// Mitsubishi GX Works2 project: fx2N_may1truc_v1.0   PLC: FX2N/FX2NC

PROGRAM MAIN
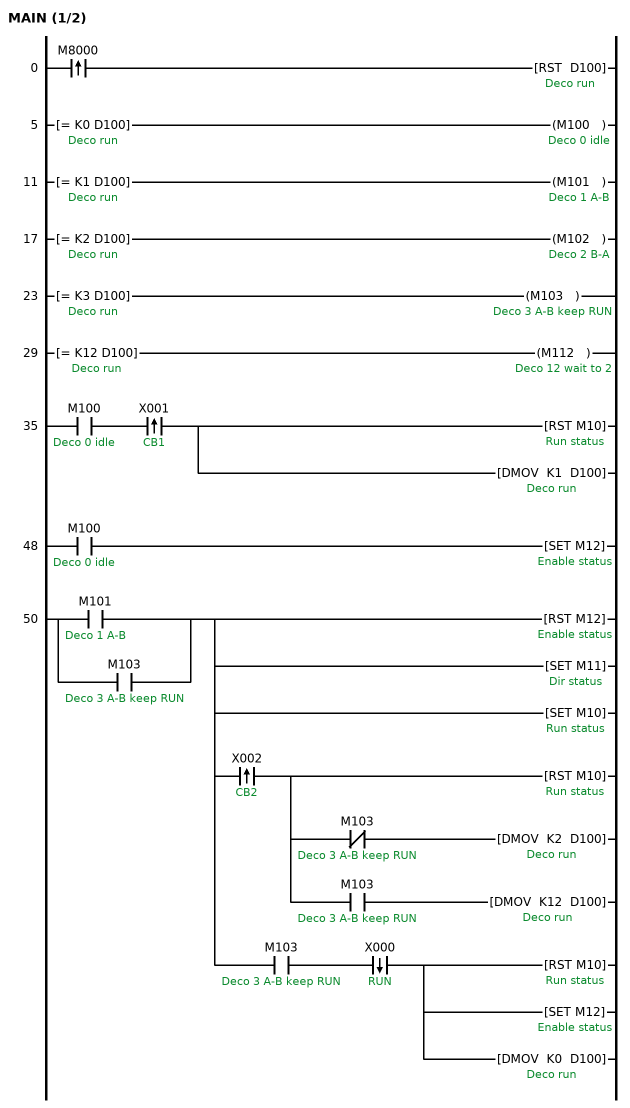
0     LDP     M8000
      RST     D100  ; Deco run
5     LD=     K0 D100  ; Deco run
      OUT     M100  ; Deco 0 idle
11    LD=     K1 D100  ; Deco run
      OUT     M101  ; Deco 1 A-B
17    LD=     K2 D100  ; Deco run
      OUT     M102  ; Deco 2 B-A
23    LD=     K3 D100  ; Deco run
      OUT     M103  ; Deco 3 A-B keep RUN
29    LD=     K12 D100  ; Deco run
      OUT     M112  ; Deco 12 wait to 2
35    LD      M100  ; Deco 0 idle
      ANDP    X001  ; CB1
      RST     M10  ; Run status
      DMOV    K1 D100
48    LD      M100  ; Deco 0 idle
      SET     M12  ; Enable status
50    LD      M101  ; Deco 1 A-B
      OR      M103  ; Deco 3 A-B keep RUN
      RST     M12  ; Enable status
      SET     M11  ; Dir status
      SET     M10  ; Run status
      MPS
      ANDP    X002  ; CB2
      RST     M10  ; Run status
      MPS
      ANI     M103  ; Deco 3 A-B keep RUN
      DMOV    K2 D100
      MPP
      AND     M103  ; Deco 3 A-B keep RUN
      DMOV    K12 D100
      MPP
      AND     M103  ; Deco 3 A-B keep RUN
      ANDF    X000  ; RUN
      RST     M10  ; Run status
      SET     M12  ; Enable status
      DMOV    K0 D100
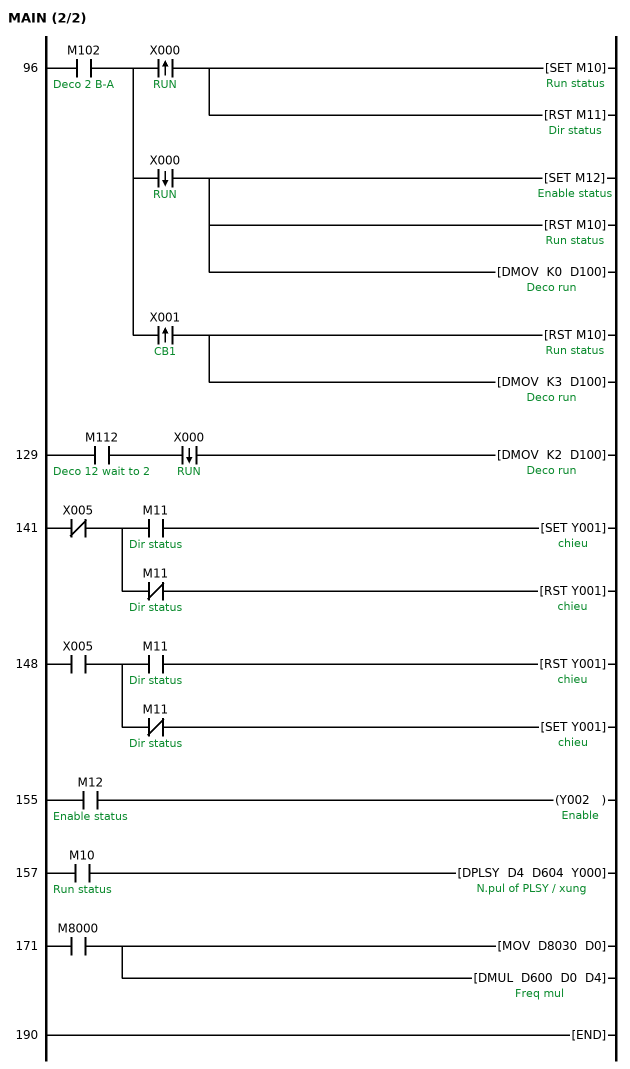
96    LD      M102  ; Deco 2 B-A
      MPS
      ANDP    X000  ; RUN
      SET     M10  ; Run status
      RST     M11  ; Dir status
      MRD
      ANDF    X000  ; RUN
      SET     M12  ; Enable status
      RST     M10  ; Run status
      DMOV    K0 D100
      MPP
      ANDP    X001  ; CB1
      RST     M10  ; Run status
      DMOV    K3 D100
129   LD      M112  ; Deco 12 wait to 2
      ANDF    X000  ; RUN
      DMOV    K2 D100
141   LDI     X005
      MPS
      AND     M11  ; Dir status
      SET     Y001  ; chieu
      MPP
      ANI     M11  ; Dir status
      RST     Y001  ; chieu
148   LD      X005
      MPS
      AND     M11  ; Dir status
      RST     Y001  ; chieu
      MPP
      ANI     M11  ; Dir status
      SET     Y001  ; chieu
155   LD      M12  ; Enable status
      OUT     Y002  ; Enable
157   LD      M10  ; Run status
      DPLSY   D4 D604 Y000  ; N.pul of PLSY / xung
171   LD      M8000
      MOV     D8030 D0
      DMUL    D600 D0 D4  ; Freq mul
190   END
END_PROGRAM

// device comments not shown above
M104  ; Deco 4
M105  ; Deco 5
M600  ; Chieu Store
